(* IEC 61131-3 sources: CodesysTest/alpha/export/PackML/OMAC/Function Blocks/UnitModeManager.pou/ActiveUnitMode.prop, 1 file *)

(* ---- Get.pm.st ---- *)
(*#-#-#-#-#-#-#-#-#-#---Declaration---#-#-#-#-#-#-#-#-#-#-#-#-#*)

VAR
END_VAR
(*#-#-#-#-#-#-#-#-#-#---Implementation---#-#-#-#-#-#-#-#-#-#-#-#-#*)

ActiveUnitMode := apum[usiActualUM];
